FUNCTION_BLOCK FB_Analogue_xcheck
VAR_INPUT
	In1:REAL;
	In2:REAL;
	Constant_window:REAL;
	Percent_window:REAL;
	Use_absolute_values:BOOL;
END_VAR
VAR_OUTPUT
	Mismatch:BOOL;
END_VAR
VAR
END_VAR

Analogue_xcheck();

METHOD Analogue_xcheck
VAR_INPUT
END_VAR
VAR_INST // added by the converter: edge detectors and wires of the graphical bodies
    _w1, _w2, _w3 : ANY;
END_VAR
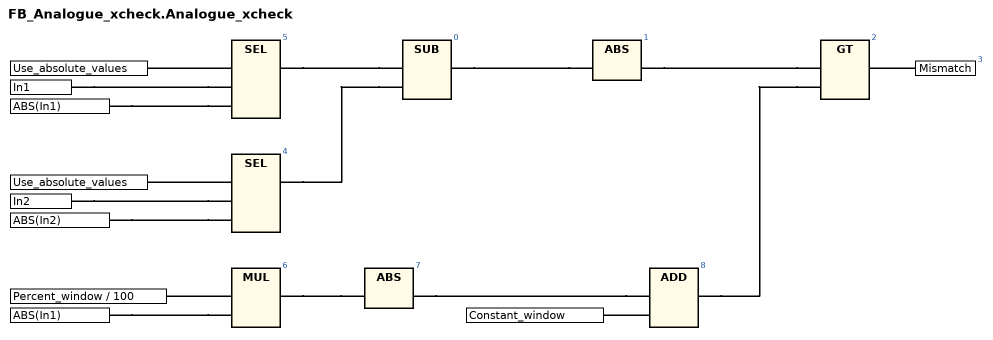
Mismatch := ABS(_w1 - _w2) > _w3;
_w2 := SEL(Use_absolute_values, In2, ABS(In2));
_w1 := SEL(Use_absolute_values, In1, ABS(In1));
_w3 := ABS((Percent_window / 100) * (ABS(In1))) + Constant_window;
END_METHOD

END_FUNCTION_BLOCK

(* stored: Version 1.1.0.1, ProductVersion 3.1.4024.0
   POU FB_Analogue_xcheck: Id {9a4723e3-eda6-405f-aaeb-af8b2fe787e5}, SpecialFunc None
   Method Analogue_xcheck: Id {cf7d7fb7-1222-4740-a074-4576c879cc4b} *)
